Staubli VAL3: getListPosition.pgx

public program getListPosition(num& x_nIndexX[], num& x_nIndexY[])
begin
  x_nIndexX=nTopX+1
  x_nIndexY=nFirst+nView+nTopY+1
end
